TYPE E_STOPREASON :
(
	StopByNone,
	StopByCommand,
	StopBySaber,
	StopByManual,
	MAX_STOPREASON
);
END_TYPE

(* stored: Version 1.1.0.1, ProductVersion 3.1.0.26
   DUT E_STOPREASON: Id {265c92cb-f90d-4512-b400-7fc9bf762399} *)
